// TwinCAT 3 PLC project Test_Project1
// ProgramVersion: 3.1.4023.0
// libraries:
//   Tc2_ControllerToolbox, * (Beckhoff Automation GmbH)
//   Tc2_Standard, * (Beckhoff Automation GmbH)
//   Tc2_System, * (Beckhoff Automation GmbH)
//   Tc3_Module, * (Beckhoff Automation GmbH)
// project tree:
//   GVLs/ GVL.TcGVL, IO.TcGVL (not stored)
//   / PID_Task.TcTTO, PlcTask.TcTTO
//   POUs/ MAIN.TcPOU
//   POUs/PID/ PRG_FB_CTRL_PID_1.TcPOU, PRG_FB_CTRL_PID_2.TcPOU, PRG_PID_CALL.TcPOU
// real-time tasks:
//   TASK PlcTask: cycle T#10ms, priority 20, ADS port 350
//   TASK PID_Task: cycle T#50000us, priority 1, ADS port 351
// I/O:
//   DEVICE Device 1 (EtherCAT), AmsNetId 5.84.189.16.2.1
//     Term 1 (EK1200) [EK1200-5000 EtherCAT Power supply (2A E-Bus)]
//       Term 2 (EL3004) [EL3004 4Ch. Ana. Input +/-10V]
//       Term 3 (EL4002) [EL4002 2Ch. Ana. Output 0-10V, 12bit]
//       Term 4 (EL9011) [EL9011 End Terminal]
// variable links:
//   Test_Project1/Test_Project1 Instance <-> Device 1 (EtherCAT)/Term 1 (EK1200)/Term 2 (EL3004)
//     PID_Task Inputs/IO.ai_tank_1_V <-> AI Standard Channel 1/Value
//     PID_Task Inputs/IO.ai_tank_2_V <-> AI Standard Channel 2/Value
//   Test_Project1/Test_Project1 Instance <-> Device 1 (EtherCAT)/Term 1 (EK1200)/Term 3 (EL4002)
//     PID_Task Outputs/IO.ao_motor_1_V <-> AO Outputs Channel 1/Analog output
//     PID_Task Outputs/IO.ao_motor_2_V <-> AO Outputs Channel 2/Analog output

CONFIGURATION Test_Project1
    RESOURCE PLC ON TwinCAT3
        TASK PID_Task(INTERVAL := T#50000us, PRIORITY := 1);
        TASK PlcTask(INTERVAL := T#10ms, PRIORITY := 20);
        PROGRAM PRG_PID_CALL WITH PID_Task : PRG_PID_CALL;
        PROGRAM MAIN WITH PlcTask : MAIN;
    END_RESOURCE
END_CONFIGURATION

// ---- GVLs/GVL.TcGVL
{attribute 'qualified_only'}
VAR_GLOBAL
	
	// To hold real value of analog input channels in V
	rAI_1 : REAL;
	rAI_2 : REAL;
	
	// To hold real value of analog output channels in V
	rAO_1 : REAL;
	rAO_2 : REAL;
	
	fSetpointValueToScope_1 : LREAL;
	fActualValueToScope_1 : LREAL;
	fOutToScope_1 : LREAL;
	fSetpointValueToScope_2 : LREAL;
	fActualValueToScope_2 : LREAL;
	fOutToScope_2 : LREAL;
END_VAR

// ---- POUs/PID/PRG_PID_CALL.TcPOU
PROGRAM PRG_PID_CALL
VAR
END_VAR



// Scale 12 bit digital voltage reading to V in range of EL3004 (0, +10)
GVL.rAI_1 := (INT_TO_REAL(IO.ai_tank_1_V)/(32767.0 - 0.0)) * 10.0;
GVL.rAI_2 := (INT_TO_REAL(IO.ai_tank_2_V)/(32767.0 - 0.0)) * 10.0;

PRG_FB_CTRL_PID_1();
PRG_FB_CTRL_PID_2();

// Unscale real V output to 12 bit digital value 
IO.ao_motor_1_V := REAL_TO_INT((GVL.rAO_1 / (10.0 - 0)) * (32767.0 - 0.0));
IO.ao_motor_2_V := REAL_TO_INT((GVL.rAO_2 / (10.0 - 0)) * (32767.0 - 0.0));

END_PROGRAM

// ---- POUs/PID/PRG_FB_CTRL_PID_1.TcPOU
PROGRAM PRG_FB_CTRL_PID_1
VAR
	fSetpointValue					: LREAL		:= 1;
	fActualValue					: LREAL;
	fManSyncValue					: LREAL;
	bSync							: BOOL;

	fOut							: LREAL;
	bHold							: BOOL;

	eMode							: E_CTRL_MODE;
	stCTRL_PID_PARAMS				: ST_CTRL_PID_PARAMS;

	eErrorId						: E_CTRL_ERRORCODES;
	bError							: BOOL;
	bARWactive						: BOOL;

	(* controller *)
	fbCTRL_PID						: FB_CTRL_PID;

	bInit							: BOOL	:= TRUE;
	fbTON							: TON;
END_VAR

IF bInit THEN
	(* init parameter struct *)
	stCTRL_PID_PARAMS.tCtrlCycleTime		:= T#50MS;
	stCTRL_PID_PARAMS.tTaskCycleTime		:= T#50MS;
	stCTRL_PID_PARAMS.fKp					:= 2.0;			(* proportional gain Kp				*)
	stCTRL_PID_PARAMS.tTn					:= T#1S;		(*  Tn								*)
	stCTRL_PID_PARAMS.tTv					:= T#200MS;		(*  Tv								*)
	stCTRL_PID_PARAMS.tTd					:= T#100MS;		(*  Td								*)
	stCTRL_PID_PARAMS.fOutMaxLimit			:= 7;			(* maximum output limit				*)
	stCTRL_PID_PARAMS.fOutMinLimit			:= 0;			(* minimum output limit				*)

	(* set the mode to ACTIVE --> normal operation *)
	eMode := eCTRL_MODE_ACTIVE;

	(* reset the init flag *)
	bInit := FALSE;
END_IF


(* copy var to scope var *)
GVL.fSetpointValueToScope_1 	:= fSetpointValue;
GVL.fActualValueToScope_1 	:= fActualValue;

fActualValue := GVL.rAI_1;

(* call controller *)
fbCTRL_PID(		fSetpointValue		:= fSetpointValue,
				fActualValue		:= fActualValue,
				fManSyncValue		:= fManSyncValue,
				bSync				:= bSync,
				eMode				:= eMode,
				bHold				:= bHold,
				stParams			:= stCTRL_PID_PARAMS,
				fOut				=> fOut,
				bARWactive			=> bARWactive,
				eErrorId			=> eErrorId,
				bError				=> bError
				);

GVL.rAO_1 := fOut;

(* copy var to scope var *)
GVL.fOutToScope_1 := fOut;

END_PROGRAM

// ---- POUs/PID/PRG_FB_CTRL_PID_2.TcPOU
PROGRAM PRG_FB_CTRL_PID_2
VAR
	fSetpointValue					: LREAL		:= 1;
	fActualValue					: LREAL;
	fManSyncValue					: LREAL;
	bSync							: BOOL;

	fOut							: LREAL;
	bHold							: BOOL;

	eMode							: E_CTRL_MODE;
	stCTRL_PID_PARAMS				: ST_CTRL_PID_PARAMS;

	eErrorId						: E_CTRL_ERRORCODES;
	bError							: BOOL;
	bARWactive						: BOOL;

	(* controller *)
	fbCTRL_PID						: FB_CTRL_PID;

	bInit							: BOOL	:= TRUE;
	fbTON							: TON;
END_VAR

IF bInit THEN
	(* init parameter struct *)
	stCTRL_PID_PARAMS.tCtrlCycleTime		:= T#50MS;
	stCTRL_PID_PARAMS.tTaskCycleTime		:= T#50MS;
	stCTRL_PID_PARAMS.fKp					:= 2.0;			(* proportional gain Kp				*)
	stCTRL_PID_PARAMS.tTn					:= T#1S;		(*  Tn								*)
	stCTRL_PID_PARAMS.tTv					:= T#200MS;		(*  Tv								*)
	stCTRL_PID_PARAMS.tTd					:= T#100MS;		(*  Td								*)
	stCTRL_PID_PARAMS.fOutMaxLimit			:= 7;			(* maximum output limit				*)
	stCTRL_PID_PARAMS.fOutMinLimit			:= 0;			(* minimum output limit				*)

	(* set the mode to ACTIVE --> normal operation *)
	eMode := eCTRL_MODE_ACTIVE;

	(* reset the init flag *)
	bInit := FALSE;
END_IF


(* copy var to scope var *)
GVL.fSetpointValueToScope_2 	:= fSetpointValue;
GVL.fActualValueToScope_2 	:= fActualValue;

fActualValue := GVL.rAI_2;

(* call controller *)
fbCTRL_PID(		fSetpointValue		:= fSetpointValue,
				fActualValue		:= fActualValue,
				fManSyncValue		:= fManSyncValue,
				bSync				:= bSync,
				eMode				:= eMode,
				bHold				:= bHold,
				stParams			:= stCTRL_PID_PARAMS,
				fOut				=> fOut,
				bARWactive			=> bARWactive,
				eErrorId			=> eErrorId,
				bError				=> bError
				);

GVL.rAO_2 := fOut;

(* copy var to scope var *)
GVL.fOutToScope_2 := fOut;

END_PROGRAM

// ---- POUs/MAIN.TcPOU
PROGRAM MAIN
VAR
END_VAR

END_PROGRAM
